{attribute 'GeneratedUsingTerminal: EK1122-0000-0018'}
{attribute addProperty BoxType "EK1122-0000-0018"}
{attribute addProperty Id "RC70_VI_AES_D_BC_ECAT_xAES_A3B0707168RC70_SAFETY_Flexi_Soft_EtherCAT_GatewayFlexi_Soft_EtherCAT_Gateway_DE394EDD5"}
{attribute addProperty CRC "645804740"}
{attribute addProperty Size "73"}
{attribute addProperty Name "RC70_A2 (EK1122)"}
TYPE RC70_A2_EK1122_267E32C4 EXTENDS EK1122_1FC0878B :
STRUCT
	{attribute addProperty Name "RC70_VI (AES-D-BC-ECAT)"}
	{attribute addProperty PreviousPort "RC70_A2 (EK1122) : D"}
	{attribute addProperty SyncUnit "C70"}
	RC70_VI_AES_D_BC_ECAT_x : AES_A3B07071;
	{attribute addProperty Name "RC70_SAFETY (Flexi Soft EtherCAT Gateway)"}
	{attribute addProperty PreviousPort "RC70_A2 (EK1122) : B"}
	{attribute addProperty SyncUnit "C70"}
	RC70_SAFETY_Flexi_Soft_EtherCAT_Gateway : Flexi_Soft_EtherCAT_Gateway_DE394EDD;
END_STRUCT
END_TYPE

(* stored: Version 1.2.0.0, ProductVersion 3.1.4024.11
   DUT RC70_A2_EK1122_267E32C4: Id {ad77c991-0caa-05d9-16e8-98691984b569} *)
